{attribute 'qualified_only'}
{attribute 'strict'}
TYPE E_Message_ECS :
(
	eNoMessage := 0,
	eTooMuchECS := 1,
	eExternalLockActive := 2,
	eErrorECS := 3,
	eNoConnectionToBackend := 4,
	eWarningECS := 5
);
END_TYPE

(* stored: Version 1.1.0.1, ProductVersion 3.1.4024.9
   DUT E_Message_ECS: Id {04deb9ff-2ca8-4a20-9f9c-d2b857906a96} *)
